FUNCTION_BLOCK FB_ToggleButton
VAR_INPUT
END_VAR
VAR_OUTPUT
END_VAR
VAR
END_VAR

END_FUNCTION_BLOCK

(* stored: Version 1.1.0.1, ProductVersion 3.1.4024.12
   POU FB_ToggleButton: Id {20c11092-cf81-40f5-b982-887e95a4637e}, SpecialFunc None *)
